// TIA Portal V17 export
// export: Created 2023-05-07T12:12:11.807973Z, ExportSetting WithDefaults, DisplayName Totally Integrated Automation Portal, DisplayVersion V17, DisplayName TIA Portal Openness, DisplayVersion V17, DisplayName TIA Portal Version Control Interface, DisplayVersion V17, DisplayName TIA Portal Test Suite Advanced, DisplayVersion V17, DisplayName STEP 7 Professional, DisplayVersion V17, DisplayName SIMATIC Energy Suite, DisplayVersion V17, DisplayName STEP 7 Safety, DisplayVersion V17, DisplayName WinCC Professional, DisplayVersion V17
DATA_BLOCK "NeuroData"   // DB18
{ S7_Optimized_Access := 'TRUE' }
VERSION : 0.1
// stored: AutoNumber true, IsOnlyStoredInLoadMemory false, IsRetainMemResEnabled false, IsWriteProtectedInAS false, MemoryReserve 100
   VAR
      finish_measurment : Bool;
      disturbance : Real;
      PV : Real;
      MV : Real;
      SP : Real;
      stop_training_inw : Bool;
      stop_training_mod : Bool;
      epoka : Real;
      error_ep_m : Real;
      error_ep_i : Real;
      error_stop_m : Real;
      error_stop_i : Real;
      epoka_m : Real;
      epoka_i : Real;
      move : Bool;
      p_move : Bool;
      finish_training : Bool;
   END_VAR
BEGIN
END_DATA_BLOCK
